Staubli VAL3: refresh.pgx

program refresh()
begin
  if (nKey>=270 and nKey<=278) or use:bUseRefresh
    call refreshStatic()
    call refreshDynamic()
  else
    // refresh the Dynamic message
    if abs(clock()-nRefresh)>nTime
      call refreshDynamic()
    endIf
  endIf
end
